FUNCTION_BLOCK GetPivot
VAR_INPUT
	tNow : LREAL;
	tTotal : LREAL;
END_VAR
VAR_OUTPUT
	pivot : LREAL;
	pivotDot : LREAL;
END_VAR
VAR
	tr : LREAL;
END_VAR

//yk  归一化规划，前半段时间匀加速到0.5，后半段时间匀减速到1
tr := tNow / tTotal;

IF tr <= 0 THEN
	pivot := 0;
	pivotDot := 0;
ELSIF tr <= 0.5 THEN
	pivot := 2.0 * tr * tr;
	pivotDot := 4.0 * tr;
ELSIF tr <= 1 THEN
	pivot := -2.0 * tr * tr + 4.0 * tr - 1.0;
	pivotDot := -4.0 * tr + 4.0;
ELSE
	pivot := 1;
	pivotDot := 0;
END_IF

END_FUNCTION_BLOCK

(* stored: Version 1.1.0.1, ProductVersion 3.1.4024.2
   POU GetPivot: Id {949da76d-1643-4a29-86f8-074b26389f00}, SpecialFunc None *)
